(* Logix 5000 project; controller testing vendor 1 type 14 code 94 rev 28.11; software revision 28.03 *)

TASK MainTask (continuous, watchdog 500 ms) : MainProgram

MODULES
   Local : vendor 1 type 14 code 94 (ICP 3, rev 28.11)
END_MODULES

TYPE STRING20 :
STRUCT
   LEN : DINT;
   DATA : SINT[20];
END_STRUCT
END_TYPE

TYPE STRING500 :
STRUCT
   LEN : DINT;
   DATA : SINT[500];
END_STRUCT
END_TYPE

TYPE Test_UDT1 :
STRUCT
   dint : DINT;
   dint_ary : DINT[5];
   real : REAL;
   real_ary : REAL[5];
   bool : BOOL;
   bool_ary : BOOL[128];
END_STRUCT
END_TYPE

TYPE Test_UDT2 :
STRUCT
   timer : TIMER;
   str : STRING;
   str20_art : STRING20[10];
   udt_ary : Test_UDT1[5];
   udt : Test_UDT1;
END_STRUCT
END_TYPE

VAR_GLOBAL   (* controller tags *)
   bool_1 : BOOL;
   bool_2 : BOOL;
   bool_3 : BOOL;
   bool_alias_1 : ALIAS FOR bool_1;
   bool_ary1 : BOOL[32];
   bool_ary2 : BOOL[2048];
   dint_1 : DINT;
   dint_2 : DINT;
   dint_3 : DINT;
   dint_alias_1 : ALIAS FOR dint_1;
   dint_ary1 : DINT[5];
   dint_ary2 : DINT[200];
   int_1 : INT;
   int_2 : INT;
   int_3 : INT;
   int_alias_1 : ALIAS FOR int_1;
   int_ary1 : INT[5];
   int_ary2 : INT[200];
   real_1 : REAL;
   real_2 : REAL;
   real_3 : REAL;
   real_alias_1 : ALIAS FOR real_1;
   real_ary1 : REAL[5];
   reaL_ARY2 : REAL[200];
   sint_1 : SINT;
   sint_2 : SINT;
   sint_3 : SINT;
   sint_ary1 : SINT[5];
   sint_ary2 : SINT[200];
   str20_1 : STRING20;
   str20_ary1 : STRING20[5];
   str500_1 : STRING500;
   str500_ary1 : STRING500[10];
   str_1 : STRING;
   str_2 : STRING;
   str_3 : STRING;
   str_alias_1 : ALIAS FOR str_1;
   str_ary1 : STRING[5];
   str_ary2 : STRING[200];
   test_udt1 : Test_UDT1;
   test_udt1_ary : Test_UDT1[5];
   test_udt1b : Test_UDT1;
   test_udt2 : Test_UDT2;
   test_udt2_ary : Test_UDT2[5];
   tmr_1 : TIMER;
   tmr_2 : TIMER;
   tmr_ary1 : TIMER[20];
   udt_alias_1 : ALIAS FOR test_udt1;
END_VAR

PROGRAM MainProgram   (* main routine MainRoutine *)
VAR
   dint_1 : DINT;
   real_1 : REAL;
   udt1_1 : Test_UDT1;
END_VAR

ROUTINE MainRoutine   (* ladder *)
END_ROUTINE
END_PROGRAM
